DATA_BLOCK "ALARM"
{ S7_Optimized_Access := 'FALSE' }
VERSION : 0.1
NON_RETAIN
   STRUCT
      FAULT : Array[0..399] of Byte;
      WARN : Array[0..399] of Byte;
      EVENT : Array[0..31] of Byte;   //  Operator (ErrorList O), byte / bit = number rule
      INFO : Array[0..39] of Byte;   //  Info (ErrorList I)
   END_STRUCT;


BEGIN

END_DATA_BLOCK

